TYPE ST_ModuleStatus :
STRUCT
END_STRUCT
END_TYPE

(* stored: Version 1.1.0.1, ProductVersion 3.1.4026.17
   DUT ST_ModuleStatus: Id {88520539-6dd6-4ad2-afe2-0cd458d3645e} *)
